{attribute 'GeneratedUsingTerminal: EL3681-0000-0021'}
{attribute addProperty BoxType "EL3681-0000-0021"}
{attribute addProperty Id "SAI_InputsAT %I*SAI_Inputs_84B29FE914SAI_FeedbackAT %I*SAI_Feedback_BDBF6DA92SAI_RangeAT %Q*SAI_Range_2A187FC54WcStateAT %I*WcState_9091E0EB2InfoDataAT %I*InfoData_32EB74EA10"}
{attribute addProperty CRC "3244640063"}
{attribute addProperty Size "32"}
TYPE EL3681_C165473F EXTENDS EtcSlaveTerminalBase_947E5A46 :
STRUCT
	{attribute addProperty Name "SAI_Inputs"}
	SAI_Inputs : SAI_Inputs_84B29FE9;
	{attribute addProperty Name "SAI_Feedback"}
	SAI_Feedback : SAI_Feedback_BDBF6DA9;
	{attribute addProperty Name "SAI_Range"}
	SAI_Range : SAI_Range_2A187FC5;
	{attribute addProperty Name "WcState"}
	WcState : WcState_9091E0EB;
	{attribute addProperty Name "InfoData"}
	InfoData : InfoData_32EB74EA;
END_STRUCT
END_TYPE

(* stored: Version 1.2.0.0, ProductVersion 3.1.4024.9
   DUT EL3681_C165473F: Id {bd681285-c77f-4704-a5cb-2882d31643b6} *)
